INTERFACE RecipeSingleValueType EXTENDS RecipeValue

METHOD ParseAndAssignValue
VAR_INPUT
	value : T_MaxString;
END_VAR
END_METHOD

END_INTERFACE

(* stored: Version 1.1.0.1, ProductVersion 3.1.4024.15
   Itf RecipeSingleValueType: Id {93d5db6c-5dfd-0676-16b7-7ee123452bed}
   Method ParseAndAssignValue: Id {6f8e467b-9b1a-06de-35c4-156e8cd2d07b} *)
